RESOURCE_TYPE TEST_RES2 (* Like TEST_RES but with PUBLISH, SUBSCRIBE *)
  (* Standard: 61499-2 *)
  (* Version 0.0, 2004-06-08, JHC, Rockwell Automation *)
  (* Compiler header: package fb.rt.test; import fb.rt.net.*; import fb.rt.math.*; *)
  VAR_INPUT
    INPUT_ID : WSTRING := "225.0.0.1:1025"; (* UDP hostport for inputs *)
    OUTPUT_ID : WSTRING := "225.0.0.1:1026"; (* UDP hostport for output *)
  END_VAR
  FB_TYPES
    FB_ADD_REAL;
  END_FB_TYPES
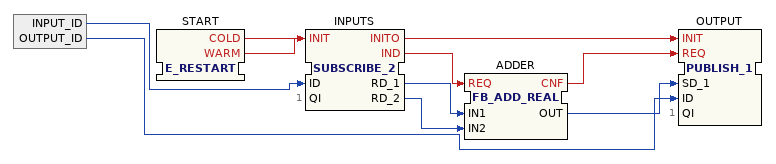
  FBS
    START : E_RESTART;
    INPUTS : SUBSCRIBE_2(QI := 1);
    ADDER : FB_ADD_REAL;
    OUTPUT : PUBLISH_1(QI := 1);
  END_FBS
  EVENT_CONNECTIONS
    START.COLD TO INPUTS.INIT;
    START.WARM TO INPUTS.INIT;
    INPUTS.INITO TO OUTPUT.INIT;
    INPUTS.IND TO ADDER.REQ;
    ADDER.CNF TO OUTPUT.REQ;
  END_CONNECTIONS
  DATA_CONNECTIONS
    INPUTS.RD_1 TO ADDER.IN1;
    INPUTS.RD_2 TO ADDER.IN2;
    ADDER.OUT TO OUTPUT.SD_1;
    INPUT_ID TO INPUTS.ID;
    OUTPUT_ID TO OUTPUT.ID;
  END_CONNECTIONS
END_RESOURCE_TYPE
